% RSLogix 500 project reject_tracking.RSS, saved by version 8.30.00.16 %
PROJECT "UNTITLED"    % processor: Bul.1763 MicroLogix 1100 Series B %

PROGRAM FILES
  LAD 2 "MAIN"  12 rungs  % Box handling program %
  LAD 240 "PE_SIMUL8R"  10 rungs  % PhotoEye (PE) state simulator %
  LAD 250 "REJSIMUL8R"  7 rungs  % Rejection simulator %

DATA FILES
  O0 OUTPUT  4 elements
  I1 INPUT  6 elements
  S2 STATUS  66 elements
  B3 BINARY  10 elements
  T4 TIMER  2 elements
  C5 COUNTER  2 elements
  R6 CONTROL  1 elements
  N7 INTEGER  1 elements
  F8 FLOAT  1 elements
  N99 FIFO  4 elements
  N199 INDEX  1 elements
  N241 INTPESML8R  3 elements
  B242 BITPESML8R  2 elements
  L251 RNGSIMUL8R  2 elements
  B252 BITSIMUL8R  1 elements

LADDER 2 "MAIN"    % Box handling program %
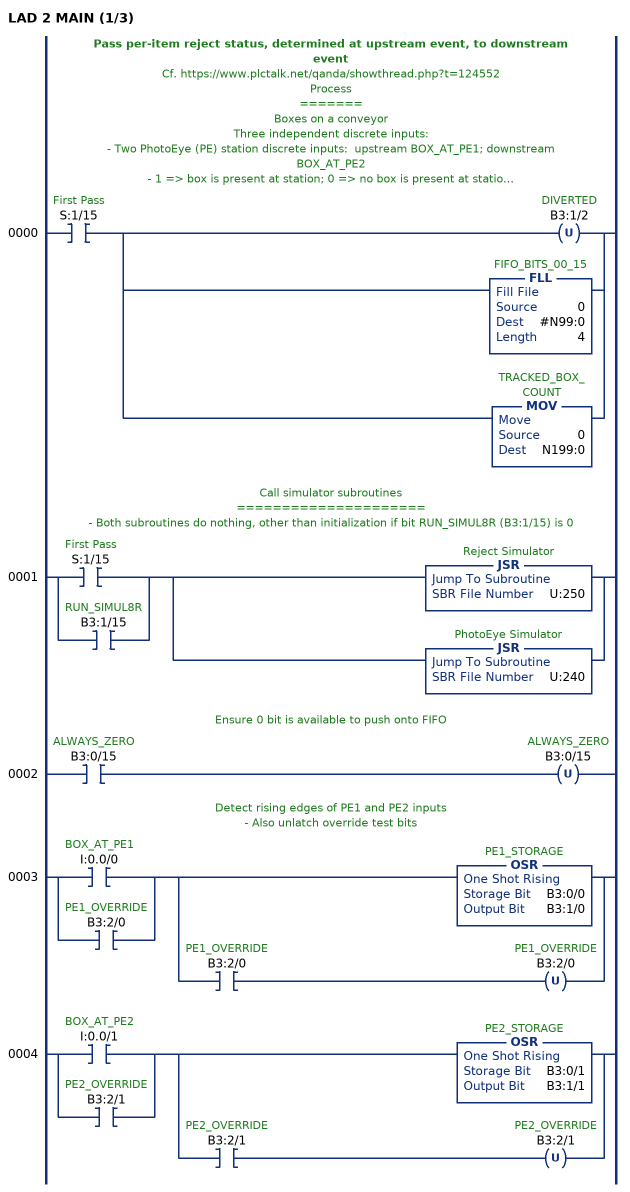
% Rung: 0 %
% TITLE: Pass per-item reject status, determined at upstream event, to downstream event %
% Cf. https://www.plctalk.net/qanda/showthread.php?t=124552
% 
% Process
% =======
% Boxes on a conveyor
% Three independent discrete inputs:
% - Two PhotoEye (PE) station discrete inputs:  upstream BOX_AT_PE1; downstream BOX_AT_PE2
%   - 1 => box is present at station; 0 => no box is present at station
% - A third discrete input REJECT_BOX_AT_PE1 determines whether a box at the upstream station either
%   - is a reject (1), and to be later diverted at PE2,
%   OR
%   - is okay (0), and not to be diverted.
% Rising edge at upstream station BOX_AT_PE1 station is where each box's {1:reject;0:okay} status is set
% - Based on the status of REJECT_BOX_AT_PE1
% When each box later generates a rising edge at downstream station BOX_AT_PE2
% - divert if box status from BOX_AT_PE1 was [reject]
% - do not divert if box status BOX_AT_PE1 was [okay]
% There will be an arbitrary number of boxes that have triggered BOX_AT_PE1 but not yet triggered BOX_AT_PE2
% - These are the only boxes this program can keep track of with the available inputs
% - The number of boxes will range from 0 to no more than approximately 10
% 
% Implementation data structures
% =========================
% Integer index TRACKED_BOX_COUNT (N199:0) is the count of tracked boxes
% - I.e boxes that have triggered BOX_AT_PE1 but not yet triggered BOX_AT_PE2
% Bit array (FIFO) in file #N99
% - Only up bits up to to N99:0/[TRACKED_BOX_COUNT-1] represent tracked boxes
% - N99 bit count = 64, whcih is much greater than the maximum possible value of TRACKED_BOX_COUNT
% - Bit value is 1 if a tracked box is a [reject] and is to be diverted at PE2
% - Bit value is 0 if a tracked box is [okay] and is not to be diverted at PE2
% - FIFO content and shifting are controlled with BSR only, not FFL/FFU
% - BSR always pushes 0-valued bit (status [okay]) at front of FIFO
%   - Which will aways be well upstream of N99:0/[TRACKED_BOX_COUNT]
% 
% Implementation events
% ==================
% At BOX_AT_PE2 rising edge
% - Pop reject/okay bit
%   - Set (or leave) DIVERTED bit state to (as) that popped bit
% - Decrement TRACKED_BOX_COUNT
% At PE1 rising edge
% - Ensure bit N99:0/[TRACKED_BOX_COUNT] has same current value as REJECT_BOX_AT_PE1
% - Increment TRACKED_BOX_COUNT
% 
% Implementation assumptions
% =======================
% There is adequate physical space between boxes, so there is exactly 1 rising edge per box at photoeyes, both at PE1, and at PE2
% No boxes are added or subtracted between PE1 and PE2, nor coffee cups blocking either PE
% 
% Initialization
% =========
% Set diverted state to 0
% - Better alternative would be detect diverter state
% Set FIFO and index to zero
% - Better alternative would be operator input of TRACKED_BOX_COUNT before starting conveyor
%   - Could also be used for resynchronization
%   - Could also set default reject/divert for any boxes past PE1 rising edge %
SOR XIC S:1/15 BST OTU B3:1/2 NXB FLL 0 #N99:0 4 NXB MOV 0 N199:0 BND EOR
%   S:1/15  "First Pass" %
%   B3:1/2  DIVERTED %
%   N99:0  FIFO_BITS_00_15 %
%   N199:0  TRACKED_BOX_COUNT %
% Rung: 1 %
% Call simulator subroutines
% =====================
% - Both subroutines do nothing, other than initialization if bit RUN_SIMUL8R (B3:1/15) is 0 %
SOR BST XIC S:1/15 NXB XIC B3:1/15 BND BST JSR U:250 NXB JSR U:240 BND EOR
%   S:1/15  "First Pass" %
%   B3:1/15  RUN_SIMUL8R %
%   U:250  "Reject Simulator" %
%   U:240  "PhotoEye Simulator" %
% Rung: 2 %
% Ensure 0 bit is available to push onto FIFO %
SOR XIC B3:0/15 OTU B3:0/15 EOR
%   B3:0/15  ALWAYS_ZERO %
% Rung: 3 %
% Detect rising edges of PE1 and PE2 inputs
% - Also unlatch override test bits %
SOR BST XIC I:0.0/0 NXB XIC B3:2/0 BND BST OSR B3:0/0 B3:1/0 NXB XIC B3:2/0 OTU B3:2/0 BND EOR
%   I:0.0/0  BOX_AT_PE1 %
%   B3:2/0  PE1_OVERRIDE %
%   B3:0/0  PE1_STORAGE %
%   B3:1/0  PE1_RISING_EDGE %
% Rung: 4 %
SOR BST XIC I:0.0/1 NXB XIC B3:2/1 BND BST OSR B3:0/1 B3:1/1 NXB XIC B3:2/1 OTU B3:2/1 BND EOR
%   I:0.0/1  BOX_AT_PE2 %
%   B3:2/1  PE2_OVERRIDE %
%   B3:0/1  PE2_STORAGE %
%   B3:1/1  PE2_RISING_EDGE %

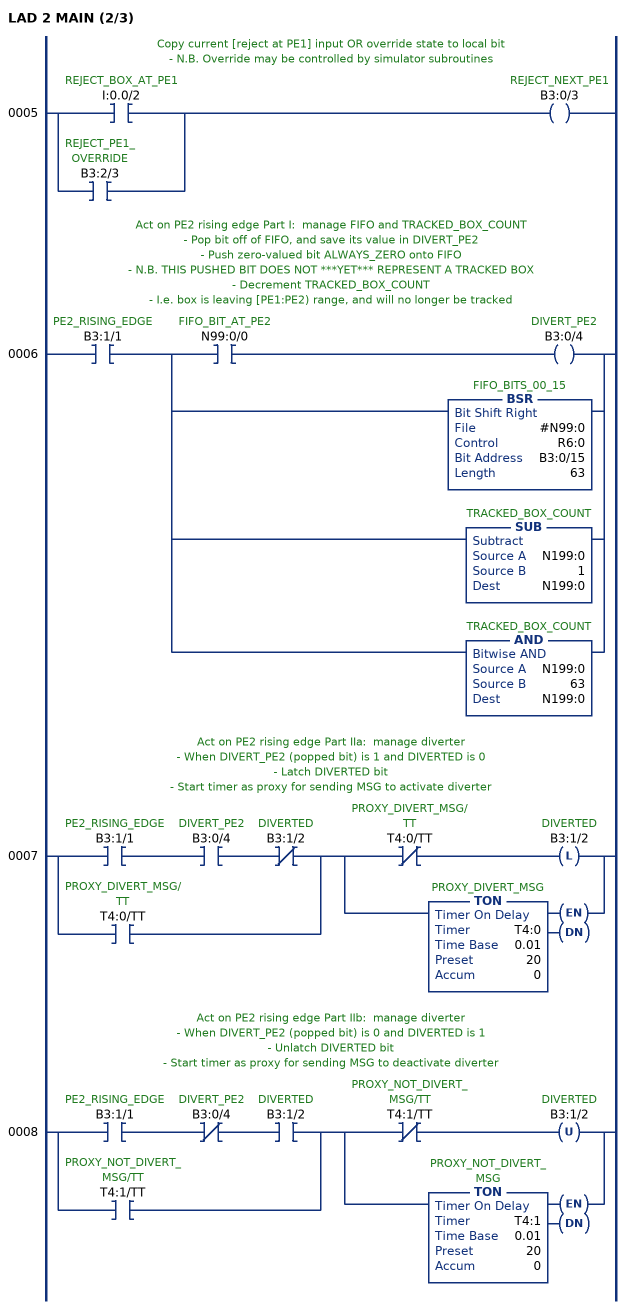
% Rung: 5 %
% Copy current [reject at PE1] input OR override state to local bit
% - N.B. Override may be controlled by simulator subroutines %
SOR BST XIC I:0.0/2 NXB XIC B3:2/3 BND OTE B3:0/3 EOR
%   I:0.0/2  REJECT_BOX_AT_PE1 %
%   B3:2/3  REJECT_PE1_OVERRIDE %
%   B3:0/3  REJECT_NEXT_PE1 %
% Rung: 6 %
% Act on PE2 rising edge Part I:  manage FIFO and TRACKED_BOX_COUNT
% - Pop bit off of FIFO, and save its value in DIVERT_PE2
% - Push zero-valued bit ALWAYS_ZERO onto FIFO
%   - N.B. THIS PUSHED BIT DOES NOT ***YET*** REPRESENT A TRACKED BOX
% - Decrement TRACKED_BOX_COUNT
%   - I.e. box is leaving [PE1:PE2) range, and will no longer be tracked %
SOR XIC B3:1/1 BST XIC N99:0/0 OTE B3:0/4 NXB BSR #N99:0 R6:0 B3:0/15 63 NXB SUB N199:0 1 N199:0 NXB AND N199:0 63 N199:0 BND EOR
%   B3:1/1  PE2_RISING_EDGE %
%   N99:0/0  FIFO_BIT_AT_PE2 %
%   B3:0/4  DIVERT_PE2 %
%   N99:0  FIFO_BITS_00_15 %
%   R6:0  ADD_FIRST_IN_AS_ZERO %
%   B3:0/15  ALWAYS_ZERO %
%   N199:0  TRACKED_BOX_COUNT %
% Rung: 7 %
% Act on PE2 rising edge Part IIa:  manage diverter
% - When DIVERT_PE2 (popped bit) is 1 and DIVERTED is 0
%   - Latch DIVERTED bit
%   - Start timer as proxy for sending MSG to activate diverter %
SOR BST XIC B3:1/1 XIC B3:0/4 XIO B3:1/2 NXB XIC T4:0/TT BND BST XIO T4:0/TT OTL B3:1/2 NXB TON T4:0 0.01 20 0 BND EOR
%   B3:1/1  PE2_RISING_EDGE %
%   B3:0/4  DIVERT_PE2 %
%   B3:1/2  DIVERTED %
%   T4:0  PROXY_DIVERT_MSG %
% Rung: 8 %
% Act on PE2 rising edge Part IIb:  manage diverter
% - When DIVERT_PE2 (popped bit) is 0 and DIVERTED is 1
%   - Unlatch DIVERTED bit
%   - Start timer as proxy for sending MSG to deactivate diverter %
SOR BST XIC B3:1/1 XIO B3:0/4 XIC B3:1/2 NXB XIC T4:1/TT BND BST XIO T4:1/TT OTU B3:1/2 NXB TON T4:1 0.01 20 0 BND EOR
%   B3:1/1  PE2_RISING_EDGE %
%   B3:0/4  DIVERT_PE2 %
%   B3:1/2  DIVERTED %
%   T4:1  PROXY_NOT_DIVERT_MSG %

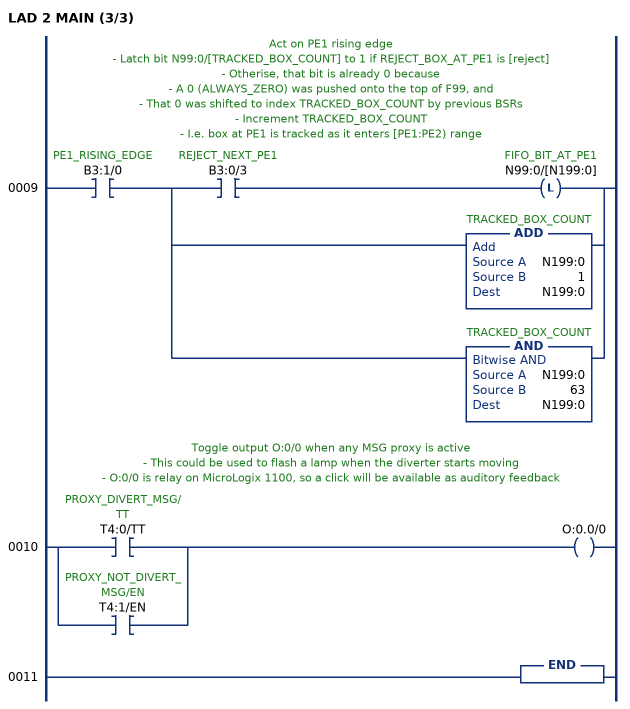
% Rung: 9 %
% Act on PE1 rising edge
% - Latch bit N99:0/[TRACKED_BOX_COUNT] to 1 if REJECT_BOX_AT_PE1 is [reject]
%   - Otherise, that bit is already 0 because
%     - A 0 (ALWAYS_ZERO) was pushed onto the top of F99, and
%     - That 0 was shifted to index TRACKED_BOX_COUNT by previous BSRs
% - Increment TRACKED_BOX_COUNT
%   - I.e. box at PE1 is tracked as it enters [PE1:PE2) range %
SOR XIC B3:1/0 BST XIC B3:0/3 OTL N99:0/[N199:0] NXB ADD N199:0 1 N199:0 NXB AND N199:0 63 N199:0 BND EOR
%   B3:1/0  PE1_RISING_EDGE %
%   B3:0/3  REJECT_NEXT_PE1 %
%   N99:0/[N199:0]  FIFO_BIT_AT_PE1 %
%   N99:0  FIFO_BITS_00_15 %
%   N199:0  TRACKED_BOX_COUNT %
% Rung: 10 %
% Toggle output O:0/0 when any MSG proxy is active
% - This could be used to flash a lamp when the diverter starts moving
% - O:0/0 is relay on MicroLogix 1100, so a click will be available as auditory feedback %
SOR BST XIC T4:0/TT NXB XIC T4:1/EN BND OTE O:0.0/0 EOR
%   T4:0  PROXY_DIVERT_MSG %
%   T4:1  PROXY_NOT_DIVERT_MSG %
% Rung: 11 %
SOR END EOR

LADDER 240 "PE_SIMUL8R"    % PhotoEye (PE) state simulator %
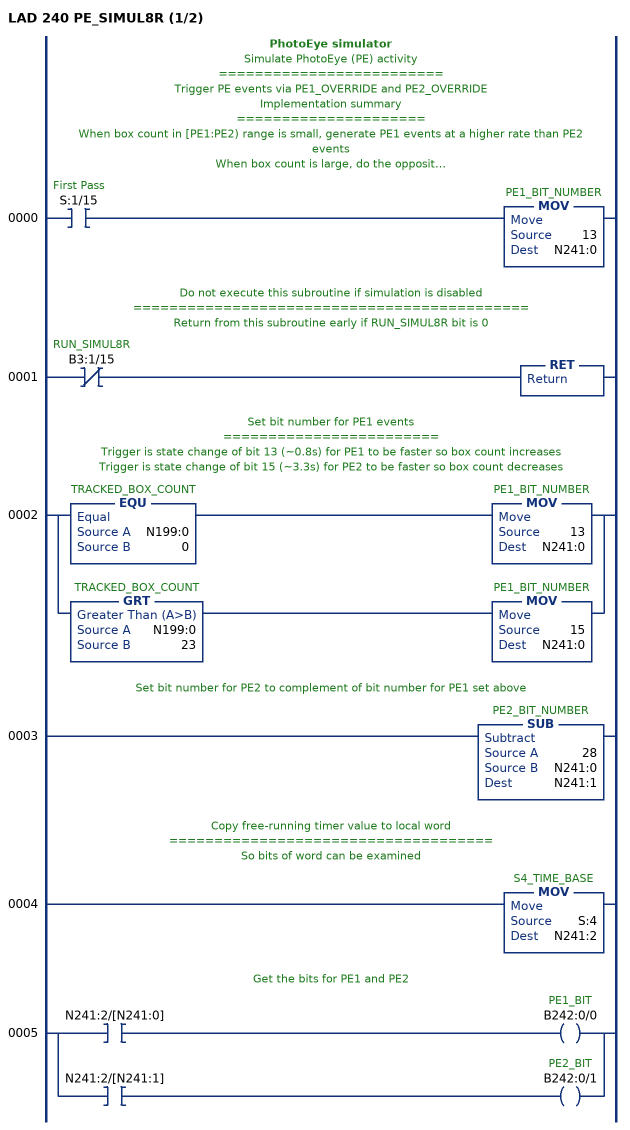
% Rung: 0 %
% TITLE: PhotoEye simulator %
% Simulate PhotoEye (PE) activity
% =========================
% Trigger PE events via PE1_OVERRIDE and PE2_OVERRIDE
% 
% Implementation summary
% =====================
% When box count in [PE1:PE2) range is small, generate PE1 events at a higher rate than PE2 events
% When box count is large, do the opposite
% 
% 
% Initialization
% =========
% Select lower bit (13 in S:4) for PE1 events %
SOR XIC S:1/15 MOV 13 N241:0 EOR
%   S:1/15  "First Pass" %
%   N241:0  PE1_BIT_NUMBER %
% Rung: 1 %
% Do not execute this subroutine if simulation is disabled
% ============================================
% Return from this subroutine early if RUN_SIMUL8R bit is 0 %
SOR XIO B3:1/15 RET EOR
%   B3:1/15  RUN_SIMUL8R %
% Rung: 2 %
% Set bit number for PE1 events
% ========================
% Trigger is state change of bit 13 (~0.8s) for PE1 to be faster so box count increases
% Trigger is state change of bit 15 (~3.3s) for PE2 to be faster so box count decreases %
SOR BST EQU N199:0 0 MOV 13 N241:0 NXB GRT N199:0 23 MOV 15 N241:0 BND EOR
%   N199:0  TRACKED_BOX_COUNT %
%   N241:0  PE1_BIT_NUMBER %
% Rung: 3 %
% Set bit number for PE2 to complement of bit number for PE1 set above %
SOR SUB 28 N241:0 N241:1 EOR
%   N241:0  PE1_BIT_NUMBER %
%   N241:1  PE2_BIT_NUMBER %
% Rung: 4 %
% Copy free-running timer value to local word
% ====================================
% So bits of word can be examined %
SOR MOV S:4 N241:2 EOR
%   S:4  "Time Base" %
%   N241:2  S4_TIME_BASE %
% Rung: 5 %
% Get the bits for PE1 and PE2 %
SOR BST XIC N241:2/[N241:0] OTE B242:0/0 NXB XIC N241:2/[N241:1] OTE B242:0/1 BND EOR
%   N241:2  S4_TIME_BASE %
%   N241:0  PE1_BIT_NUMBER %
%   B242:0/0  PE1_BIT %
%   N241:1  PE2_BIT_NUMBER %
%   B242:0/1  PE2_BIT %

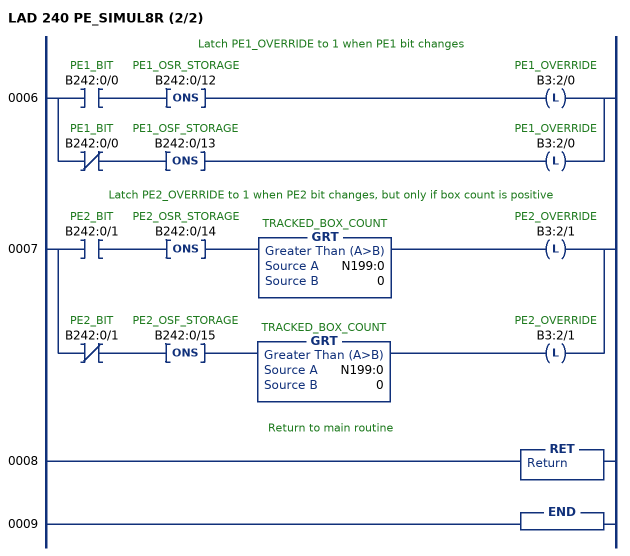
% Rung: 6 %
% Latch PE1_OVERRIDE to 1 when PE1 bit changes %
SOR BST XIC B242:0/0 ONS B242:0/12 OTL B3:2/0 NXB XIO B242:0/0 ONS B242:0/13 OTL B3:2/0 BND EOR
%   B242:0/0  PE1_BIT %
%   B242:0/12  PE1_OSR_STORAGE %
%   B3:2/0  PE1_OVERRIDE %
%   B242:0/13  PE1_OSF_STORAGE %
% Rung: 7 %
% Latch PE2_OVERRIDE to 1 when PE2 bit changes, but only if box count is positive %
SOR BST XIC B242:0/1 ONS B242:0/14 GRT N199:0 0 OTL B3:2/1 NXB XIO B242:0/1 ONS B242:0/15 GRT N199:0 0 OTL B3:2/1 BND EOR
%   B242:0/1  PE2_BIT %
%   B242:0/14  PE2_OSR_STORAGE %
%   N199:0  TRACKED_BOX_COUNT %
%   B3:2/1  PE2_OVERRIDE %
%   B242:0/15  PE2_OSF_STORAGE %
% Rung: 8 %
% Return to main routine %
SOR RET EOR
% Rung: 9 %
SOR END EOR

LADDER 250 "REJSIMUL8R"    % Rejection simulator %
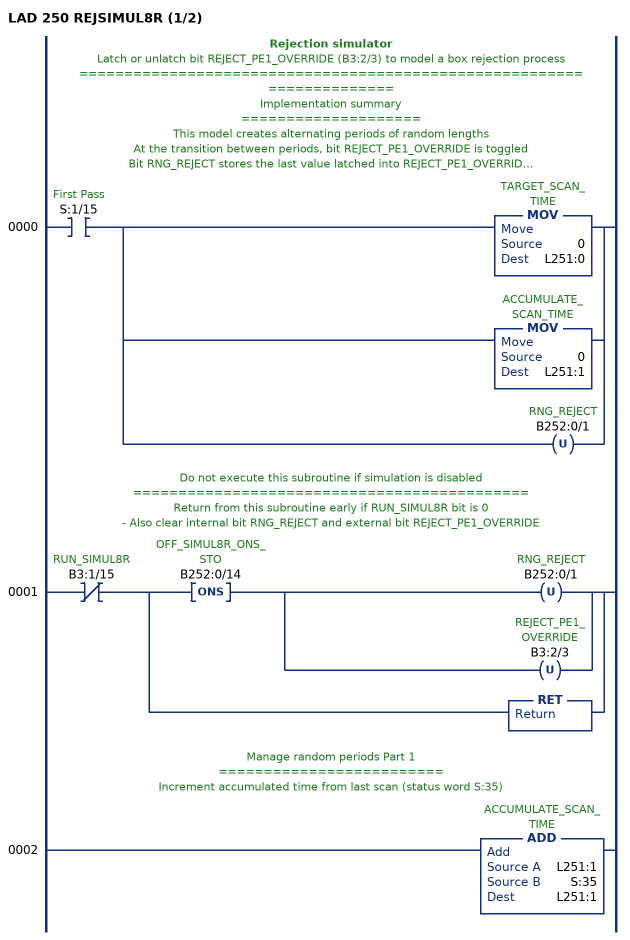
% Rung: 0 %
% TITLE: Rejection simulator %
% Latch or unlatch bit REJECT_PE1_OVERRIDE (B3:2/3) to model a box rejection process
% ======================================================================
% 
% Implementation summary
% ====================
% This model creates alternating periods of random lengths
% At the transition between periods, bit REJECT_PE1_OVERRIDE is toggled
% Bit RNG_REJECT stores the last value latched into REJECT_PE1_OVERRIDE
% 
% Initialization
% ===========
% Reset scan time variables
% Unlatch RNG_REJECT %
SOR XIC S:1/15 BST MOV 0 L251:0 NXB MOV 0 L251:1 NXB OTU B252:0/1 BND EOR
%   S:1/15  "First Pass" %
%   L251:0  TARGET_SCAN_TIME %
%   L251:1  ACCUMULATE_SCAN_TIME %
%   B252:0/1  RNG_REJECT %
% Rung: 1 %
% Do not execute this subroutine if simulation is disabled
% ============================================
% Return from this subroutine early if RUN_SIMUL8R bit is 0
% - Also clear internal bit RNG_REJECT and external bit REJECT_PE1_OVERRIDE %
SOR XIO B3:1/15 BST ONS B252:0/14 BST OTU B252:0/1 NXB OTU B3:2/3 BND NXB RET BND EOR
%   B3:1/15  RUN_SIMUL8R %
%   B252:0/14  OFF_SIMUL8R_ONS_STO %
%   B252:0/1  RNG_REJECT %
%   B3:2/3  REJECT_PE1_OVERRIDE %
% Rung: 2 %
% Manage random periods Part 1
% =========================
% Increment accumulated time from last scan (status word S:35) %
SOR ADD L251:1 S:35 L251:1 EOR
%   L251:1  ACCUMULATE_SCAN_TIME %
%   S:35  LAST_SCAN_100US  "Last 1 ms Scan Time" %

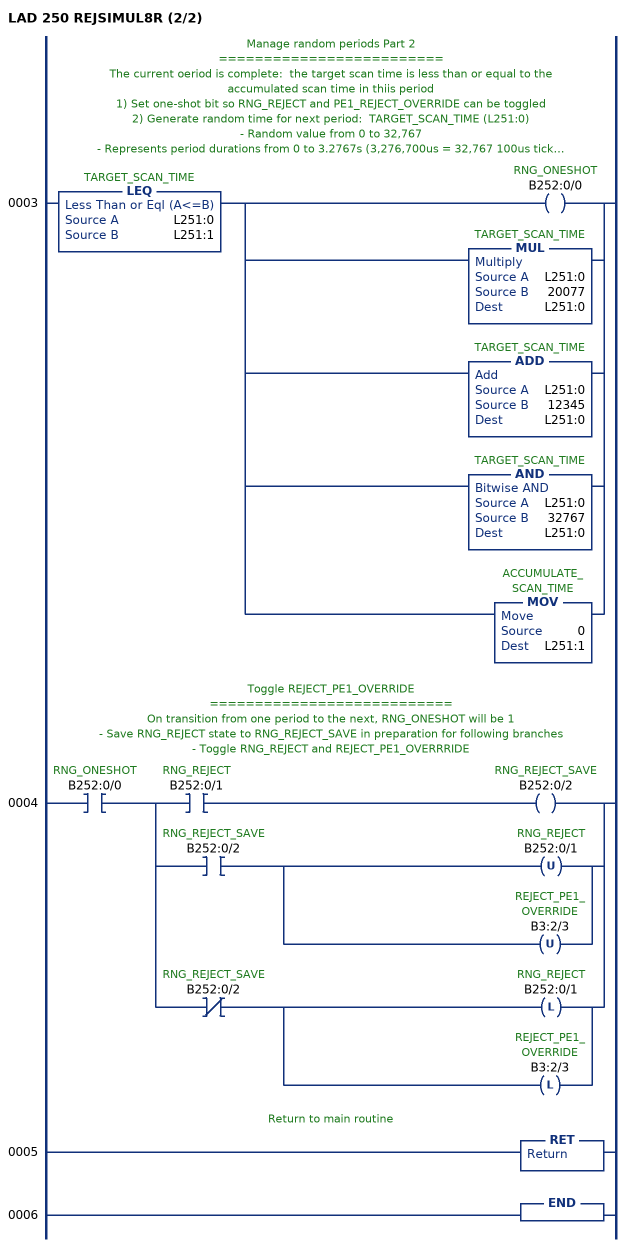
% Rung: 3 %
% Manage random periods Part 2
% =========================
% The current oeriod is complete:  the target scan time is less than or equal to the accumulated scan time in thiis period
% 
% 1) Set one-shot bit so RNG_REJECT and PE1_REJECT_OVERRIDE can be toggled
% 2) Generate random time for next period:  TARGET_SCAN_TIME (L251:0)
%      - Random value from 0 to 32,767
%      - Represents period durations from 0 to 3.2767s (3,276,700us = 32,767 100us tick)
% 3) Reset accumulated time to zero:  ACCUMULATE_SCAN_TIME (L251:1)
%      - Will be increased by S:35 in previous rung once per scan. %
SOR LEQ L251:0 L251:1 BST OTE B252:0/0 NXB MUL L251:0 20077 L251:0 NXB ADD L251:0 12345 L251:0 NXB AND L251:0 32767 L251:0 NXB MOV 0 L251:1 BND EOR
%   L251:0  TARGET_SCAN_TIME %
%   L251:1  ACCUMULATE_SCAN_TIME %
%   B252:0/0  RNG_ONESHOT %
% Rung: 4 %
% Toggle REJECT_PE1_OVERRIDE
% ===========================
% On transition from one period to the next, RNG_ONESHOT will be 1
% - Save RNG_REJECT state to RNG_REJECT_SAVE in preparation for following branches
% - Toggle RNG_REJECT and REJECT_PE1_OVERRRIDE %
SOR XIC B252:0/0 BST XIC B252:0/1 OTE B252:0/2 NXB XIC B252:0/2 BST OTU B252:0/1 NXB OTU B3:2/3 BND NXB XIO B252:0/2 BST OTL B252:0/1 NXB OTL B3:2/3 BND BND EOR
%   B252:0/0  RNG_ONESHOT %
%   B252:0/1  RNG_REJECT %
%   B252:0/2  RNG_REJECT_SAVE %
%   B3:2/3  REJECT_PE1_OVERRIDE %
% Rung: 5 %
% Return to main routine %
SOR RET EOR
% Rung: 6 %
SOR END EOR

OTHER DOCUMENTED ADDRESSES
  B3:0/2  DIVERTED_STORE
  B242:1/12  PE1_OSR
  B242:1/13  PE1_OSF
  B242:1/14  PE2_OSR
  B242:1/15  PE2_OSF
  C5:0  PE1_OVERRIDE_COUNT
  C5:1  PE2_OVERRIDE_COUNT
  L99:0  FIRST_32
  L99:0/0  NEXT_PE2_DIVERT_BIT
  L99:0/[N199:0]  NEXT_PE1_REJECT_BIT
  L99:1  SECOND_32
  L99:2  ZERO_BIT_SOURCE
  N99:1  FIFO_BITS_16_31
  N99:2  FIFO_BITS_32_47
  N99:3  FIFO_BITS_48_63

DATA TABLE (non-zero values as saved)
DATA T4
% .PRE .ACC %
% T4:0 % 20 0
% T4:1 % 20 0
DATA C5
% .PRE .ACC %
% C5:0 % 100 0
% C5:1 % 100 0
DATA R6
% .LEN .POS %
% R6:0 % 63 0
